Staubli VAL3: cycle_start.pgx

program cycle_start()
  local num l_nID
  local num l_nId
  local string l_sName
begin
  //
  // Start the cycle
  //
  call processList:getCycle(l_sName,l_nID,l_nID,0,1)
  if l_sName!=""
    logMsg("[KERNEL] PLC:Start Cycle")
    nToSuperV=0
    wait(nToSuperV==-1)
  endIf
end
